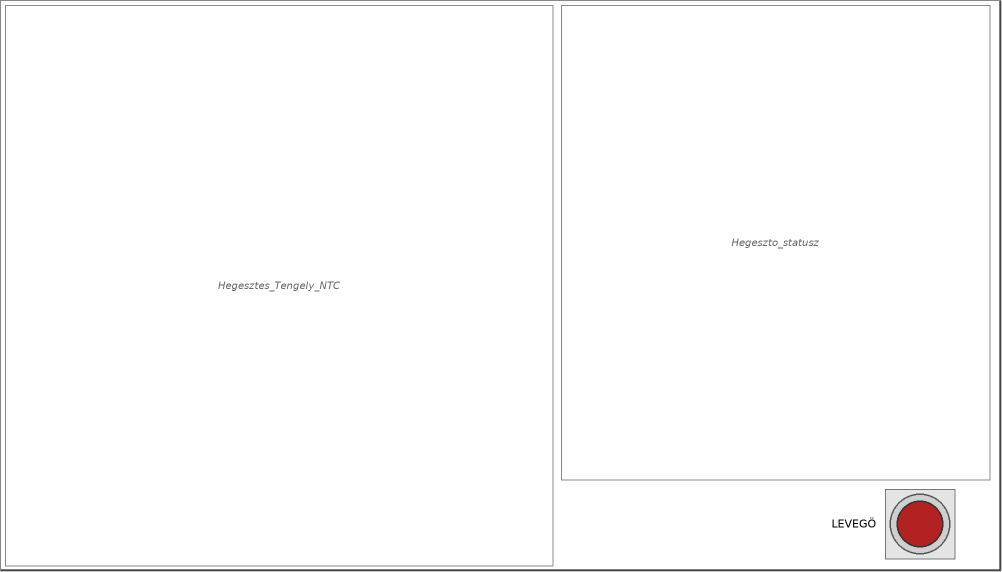
VISUALIZATION Hegesztok  // 1002x572
    Rectangle (0,0 1000x570)
    TabControl (5,5 548x561), frame switch variable: GVL.iTengelyLapozo
        shows Hegesztes_Tengely_NTC()
        shows Hegesztes_Tengely_Pt1000()
        shows Hegesztes_Karbantartas()
        [0]: TabTitle=NTC oldal
        [1]: TabTitle=Pt1000 oldal
        [2]: TabTitle=Elekróda karbantartás
    Group (824,489 131x70)
        PushSwitch (61,0 70x70), variable: MAIN.bLevego, behaviour: TOGGLE, style: Switch-PushSwitch-Red
        Label (0,20 55x30), "LEVEGÖ"
    TabControl (561,5 429x475)
        shows Hegeszto_statusz()
        shows Hegesztofej_IOk()
        shows Pt1000_oldali_kamera()
        [0]: TabTitle=Hegesztö státusz
        [1]: TabTitle=Hegesztöfej I/O-k
        [2]: TabTitle=Pt oldali kamera
END_VISUALIZATION

(* stored: Version 1.1.0.1, ProductVersion 3.1.4024.11
   Visu Hegesztok: Id {bd065c67-ad32-478d-b794-2c31173ddfd9} *)
